{attribute 'GeneratedUsingTerminal: EL9221-4030-0018'}
{attribute addProperty BoxType "EL9221-4030-0018"}
{attribute addProperty Id "ControlAT %Q*Control_534FEB192"}
{attribute addProperty CRC "16861492"}
{attribute addProperty Size "2"}
TYPE OCP_Outputs_01014934 EXTENDS OutputBase_10CEE7DE :
STRUCT
	{attribute addProperty Name "Control"}
	Control AT %Q* : Control_534FEB19;
END_STRUCT
END_TYPE

(* stored: Version 1.2.0.0, ProductVersion 3.1.4024.9
   DUT OCP_Outputs_01014934: Id {711ad214-9a17-4d71-b08c-6c1400d33df9} *)
